INTERFACE I_MoveAbsolute

METHOD MoveAbsolute
VAR_INPUT
    Execute     : BOOL;
    Position	: LREAL;
    Velocity	: LREAL;
    Acceleration	: LREAL := 0.0;
    Deceleration	: LREAL := 0.0;
    Jerk	: LREAL := 0.0;
    BufferMode	: MC_BufferMode := MC_BufferMode.MC_Aborting;
END_VAR
END_METHOD

PROPERTY MoveAbsoluteAborted : BOOL
GET
END_GET
END_PROPERTY

PROPERTY MoveAbsoluteActive : BOOL
GET
END_GET
END_PROPERTY

PROPERTY MoveAbsoluteBusy : BOOL
GET
END_GET
END_PROPERTY

PROPERTY MoveAbsoluteDone : BOOL
GET
END_GET
END_PROPERTY

PROPERTY MoveAbsoluteError : BOOL
GET
END_GET
END_PROPERTY

PROPERTY MoveAbsoluteErrorID : UDINT
GET
END_GET
END_PROPERTY

END_INTERFACE

(* stored: Version 1.1.0.1
   Itf I_MoveAbsolute: Id {7b52c23d-d549-4d14-b715-d0e842580738}
   Method MoveAbsolute: Id {6ca50ed1-00a4-4a5f-9fc0-b477fbaad08d}
   Property MoveAbsoluteAborted: Id {3cbc255c-75e9-4ad4-a183-f5d79abd7d2b}
   Get Get: Id {e3e0c1b9-421e-4378-a6f0-95d48d7a619d}
   Property MoveAbsoluteActive: Id {aa5e4d9b-53b9-487d-aa20-131cb555a892}
   Get Get: Id {0e48ad5c-2521-41b7-88a3-39e827f8d022}
   Property MoveAbsoluteBusy: Id {695fcc39-186c-4331-9098-de70b03fd558}
   Get Get: Id {b5ea92b2-4cd9-455c-b6ae-9da22a8b84d9}
   Property MoveAbsoluteDone: Id {9ba59f72-6f0b-4c7b-9343-7af113119a76}
   Get Get: Id {a34a1cda-ed04-489a-89f2-807a4c2bf78a}
   Property MoveAbsoluteError: Id {34282d73-6471-48bf-87a6-c6af02a98f04}
   Get Get: Id {31231d6b-76fb-4529-8c95-187eb6dd1fec}
   Property MoveAbsoluteErrorID: Id {4ae355cc-eee9-4dbf-994c-6409e14defe6}
   Get Get: Id {978b51ff-6054-4e34-8e91-21c1296fde0b} *)
